TYPE TcoGenericInterpolatorHwInputs :
STRUCT
	iToPlc AT %I* : NCTOPLC_NCICHANNEL_REF;
END_STRUCT
END_TYPE

(* stored: Version 1.1.0.1, ProductVersion 3.1.4024.12
   DUT TcoGenericInterpolatorHwInputs: Id {f6dd5014-c3e3-41bc-be15-ec353d61fa37} *)
